{attribute 'pack_mode' := '1'}
(*already a built in struct called ST_AxisStatus so leaving this as AxisStatus instead*)
TYPE AxisStatus:
STRUCT
    actPos		: LREAL;	(* Actual position in mm. *)
    actVel		: LREAL;	(* Actual velocity in mm/sec. *)
    setAcc		: LREAL;	(* Set acceleration in mm/sec^2.*)
	enabled		: BOOL;		(* Is the axis enabled? *)
	brakeSet	: BOOL;		(* Is the brake engaged? *)
    lowLimit	: BOOL;		(* Low limit switch tripped? *)
	highLimit	: BOOL; 	(* High limit switch tripped? *)
	isHomed		: BOOL; 	(* Has the axis been homed? *)
	errorID		: UDINT; 	(* Axis error code. *)
    icTemp	: LREAL; 	    (* Temperature of motor controller IC, Celsius. *)
END_STRUCT
END_TYPE

(* stored: Version 1.1.0.1, ProductVersion 3.1.4022.18
   DUT AxisStatus: Id {d3960a1d-410e-4213-835a-7744e6881da9} *)
